FUNCTION_BLOCK FIELDBUS_WORD_TO_SIGNAL_SCALED (* Mirrors IN->OUT if Signal Valid, with scaling *)
  (* Standard: 61499-1; Description: Copyright (c) 2026 HR Agrartechnik GmbH This program and the accompanying materials are made available under the terms of the Eclipse Public License 2.0 which is available at https://www.eclipse.org/legal/epl-2.0/ SPDX-License-Identifier: EPL-2.0 *)
  (* Version 1.0, 2026-05-31, Franz Höpfinger, HR Agrartechnik GmbH *)
  PACKAGE logiBUS::signalprocessing::fieldbus;
  IMPORT eclipse4diac::signalprocessing::FIELDBUS_SIGNAL::NOT_AVAILABLE_WM;
  IMPORT eclipse4diac::signalprocessing::FIELDBUS_SIGNAL::VALID_SIGNAL_W;
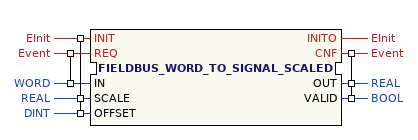
  EVENT_INPUT
    INIT : EInit WITH SCALE, OFFSET; (* Init Request *)
    REQ WITH IN; (* Normal Execution Request *)
  END_EVENT
  EVENT_OUTPUT
    INITO : EInit; (* Init Confirmation *)
    CNF WITH OUT, VALID; (* Execution Confirmation *)
  END_EVENT
  VAR_INPUT
    IN : WORD := NOT_AVAILABLE_WM; (* Input *)
    SCALE : REAL := REAL#1.0; (* Scaling factor *)
    OFFSET : DINT := DINT#0; (* Offset added after scaling *)
  END_VAR
  VAR_OUTPUT
    OUT : REAL := REAL#0.0; (* Output Scaled *)
    VALID : BOOL := FALSE; (* TRUE if Signal is VALID *)
  END_VAR
  EC_STATES
    INIT : INIT -> INITO;
    REQ : REQ -> CNF;
  END_STATES
  ALGORITHM INIT IN ST:

  END_ALGORITHM
  ALGORITHM REQ IN ST: (* Executed algorithm *)
IF (WORD_TO_UINT(IN) <= WORD_TO_UINT(VALID_SIGNAL_W)) THEN
	OUT := UINT_TO_REAL(WORD_TO_UINT(IN)) * SCALE + DINT_TO_REAL(OFFSET);
	VALID := BOOL#TRUE;
ELSE
	OUT := REAL#0.0;
	VALID := BOOL#FALSE;
END_IF;
  END_ALGORITHM
END_FUNCTION_BLOCK
